// TwinCAT 3 PLC project Plc
// Title: InvokeCSharp
// Company: Inxton
// Author: Inxton-Dev-Team
// ProjectVersion: 0.0.0.0
// ProgramVersion: 3.1.4023.0
// libraries:
//   Tc2_Standard, * (Beckhoff Automation GmbH)
//   Tc2_System, * (Beckhoff Automation GmbH)
//   Tc3_Module, * (Beckhoff Automation GmbH)
//   TcoCore, 0.5.0.829 (Vortex.Library)
// project tree:
//   / PlcTask.TcTTO (not stored)
//   POUs/ App.TcPOU, MAIN.TcPOU (not stored)
// real-time tasks:
//   TASK PlcTask: cycle T#10ms, priority 20, ADS port 350

// ---- POUs/App.TcPOU


FUNCTION_BLOCK App EXTENDS TcoCore.TcoContext
VAR
	Increment: REAL;
//	Invoke_C_Sharp: TcoCore.TcoRemoteTask(THIS^);
END_VAR

(*~
	<docu>
		<summary>
			Main method of the TcoContext. This is the entry point of any control logic that belongs to this context. 
			The call of this method is ensured by calling the <c>InstanceName.Run()</c> method, and it must not be called explicitly.
			This method is abstract, and it must be overridden in derived block.
		</summary>
	</docu>
~*)
METHOD PROTECTED  Main
//Invoke_C_Sharp();

Increment:= Increment + 1;

IF (REAL_TO_INT(Increment) MOD 500) = 0 THEN
	
//	Invoke_C_Sharp.Invoke();

END_IF
END_METHOD

END_FUNCTION_BLOCK
